% RSLogix 500 project Problom 4 lab 1 auto.RSS, saved by version 8.40.00.08 %
PROJECT "UNTITLED"    % processor: type code 33 %

PROGRAM FILES
  LAD 2   8 rungs

DATA FILES
  O0 OUTPUT  70 elements
  I1 INPUT  66 elements
  S2 STATUS  164 elements
  B3 BINARY  1 elements
  T4 TIMER  1 elements
  C5 COUNTER  1 elements
  R6 CONTROL  1 elements
  N7 INTEGER  1 elements
  F8 FLOAT  1 elements

LADDER 2
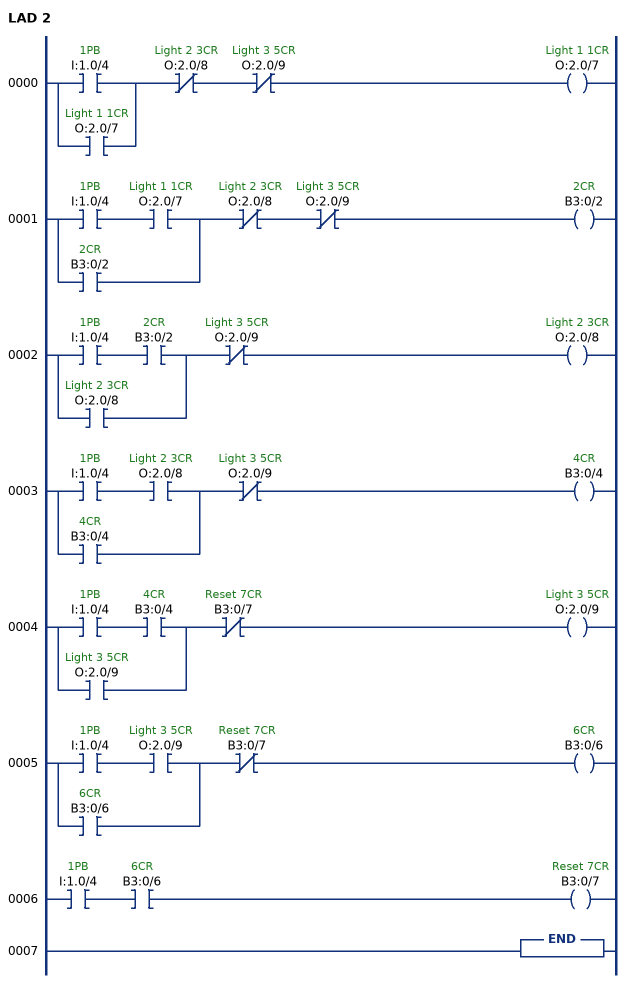
% Rung: 0 %
SOR BST XIC I:1.0/4 NXB XIC O:2.0/7 BND XIO O:2.0/8 XIO O:2.0/9 OTE O:2.0/7 EOR
%   I:1.0/4  1PB %
%   O:2.0/7  1CR  "Light 1" %
%   O:2.0/8  3CR  "Light 2" %
%   O:2.0/9  5CR  "Light 3" %
% Rung: 1 %
SOR BST XIC I:1.0/4 XIC O:2.0/7 NXB XIC B3:0/2 BND XIO O:2.0/8 XIO O:2.0/9 OTE B3:0/2 EOR
%   I:1.0/4  1PB %
%   O:2.0/7  1CR  "Light 1" %
%   B3:0/2  2CR %
%   O:2.0/8  3CR  "Light 2" %
%   O:2.0/9  5CR  "Light 3" %
% Rung: 2 %
SOR BST XIC I:1.0/4 XIC B3:0/2 NXB XIC O:2.0/8 BND XIO O:2.0/9 OTE O:2.0/8 EOR
%   I:1.0/4  1PB %
%   B3:0/2  2CR %
%   O:2.0/8  3CR  "Light 2" %
%   O:2.0/9  5CR  "Light 3" %
% Rung: 3 %
SOR BST XIC I:1.0/4 XIC O:2.0/8 NXB XIC B3:0/4 BND XIO O:2.0/9 OTE B3:0/4 EOR
%   I:1.0/4  1PB %
%   O:2.0/8  3CR  "Light 2" %
%   B3:0/4  4CR %
%   O:2.0/9  5CR  "Light 3" %
% Rung: 4 %
SOR BST XIC I:1.0/4 XIC B3:0/4 NXB XIC O:2.0/9 BND XIO B3:0/7 OTE O:2.0/9 EOR
%   I:1.0/4  1PB %
%   B3:0/4  4CR %
%   O:2.0/9  5CR  "Light 3" %
%   B3:0/7  7CR  "Reset" %
% Rung: 5 %
SOR BST XIC I:1.0/4 XIC O:2.0/9 NXB XIC B3:0/6 BND XIO B3:0/7 OTE B3:0/6 EOR
%   I:1.0/4  1PB %
%   O:2.0/9  5CR  "Light 3" %
%   B3:0/6  6CR %
%   B3:0/7  7CR  "Reset" %
% Rung: 6 %
SOR XIC I:1.0/4 XIC B3:0/6 OTE B3:0/7 EOR
%   I:1.0/4  1PB %
%   B3:0/6  6CR %
%   B3:0/7  7CR  "Reset" %
% Rung: 7 %
SOR END EOR
